{attribute 'OPC.UA.DA' := '0'}
TYPE PowermeterSensor :
STRUCT
	Name : STRING;
	Wavelength : UINT;
	Attenuation : UINT;
END_STRUCT
END_TYPE

(* stored: Version 1.1.0.1, ProductVersion 3.1.4024.4
   DUT PowermeterSensor: Id {029b2220-b9e0-4b96-971f-264f541b6e26} *)
